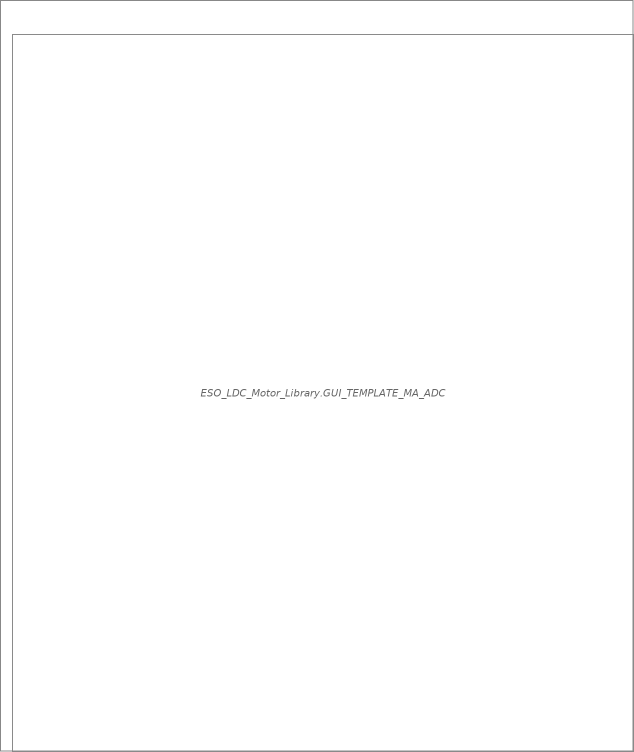
VISUALIZATION adc1  // 634x752
    Frame (12,34 622x718)
        shows ESO_LDC_Motor_Library.GUI_TEMPLATE_MA_ADC(m_DeviceName := 'ADC1', m_Instance := MAIN.adc1)
END_VISUALIZATION

(* stored: Version 1.1.0.1, ProductVersion 3.1.4024.3
   Visu adc1: Id {a411c465-72fe-4afb-8923-37374b5fa0dd} *)
